FUNCTION_BLOCK SetAllOverrideVisitor IMPLEMENTS I_ModuleVisitor, I_ComponentVisitor
VAR
	ipOverride : I_Override;
	_Override  : LREAL;
END_VAR

METHOD Set
VAR_INPUT
	Module	 : I_Module;
	Override : LREAL;
END_VAR
_Override := Override;
Module.Accept(THIS^);
IF __QUERYINTERFACE(Module, ipOverride) THEN
	ipOverride.Override := _Override;
END_IF
END_METHOD

METHOD VisitComponent
VAR_INPUT
	Component : I_Component;
END_VAR
IF __QUERYINTERFACE(Component, ipOverride) THEN
	ipOverride.Override := _Override;
END_IF
END_METHOD

METHOD VisitModule
VAR_INPUT
	Module : I_Module;
END_VAR
Module.Components.Accept(THIS^);
Module.Modules.Accept(THIS^);
IF __QUERYINTERFACE(Module, ipOverride) THEN
	ipOverride.Override := _Override;
END_IF
END_METHOD

END_FUNCTION_BLOCK

(* stored: Version 1.1.0.1, ProductVersion 3.1.4026.18
   POU SetAllOverrideVisitor: Id {3a260527-c935-473e-9804-23158d399a94}, SpecialFunc None
   Method Set: Id {3fa54dce-4562-41a3-9198-926dbe041fe1}
   Method VisitComponent: Id {5c4322d3-4089-451e-9e28-f45e18e4b32b}
   Method VisitModule: Id {86465fc1-b94b-47ca-a1b4-7683efffc6f1} *)
